// TwinCAT 3 PLC project EPS_Tests
// ProgramVersion: 3.1.4020.5
// libraries:
//   EPS, * (SLAC)
//   Tc2_BABasic, * (Beckhoff Automation GmbH)
//   Tc2_Standard, * (Beckhoff Automation GmbH)
//   Tc2_System, * (Beckhoff Automation GmbH)
//   Tc3_Module, * (Beckhoff Automation GmbH)
//   TcUnit, * (www.tcunit.org)
// project tree:
//   / PlcTask.TcTTO
//   POUs/Fixtures/AmphosMRC/ F_AmphosMRC_Error.TcPOU
//   POUs/Fixtures/BaseplateChiller/ F_BaseplateChiller_Error.TcPOU
//   POUs/Fixtures/DumpChiller/ F_DumpChiller_Error.TcPOU
//   POUs/Fixtures/Laser/ F_Laser_Error.TcPOU, F_LaserSetpoints.TcPOU
//   POUs/Fixtures/ChillerLoop/ F_ChillerLoop_Error.TcPOU
//   POUs/Fixtures/LeakMonitor/ F_LeakBoundaries.TcPOU, F_LeakMonitor_LIR_1.TcPOU, F_LeakMonitor_LIR_2.TcPOU, F_LeakMonitor_LOCO_2.TcPOU, F_LeakMonitor_LOTAO_2.TcPOU, F_LeakMonitor_LOTNL_1.TcPOU, F_LeakMonitor_LOTAO_1.TcPOU, F_LeakMonitor_LOCO_1.TcPOU, F_LeakMonitor_LOTNL_2.TcPOU, F_LeakMonitor_LUT_1.TcPOU, F_LeakMonitor_LUT_2.TcPOU
//   POUs/Fixtures/TemperatureMonitor/ F_TemperatureMonitorSetpoints.TcPOU, F_TemperatureMonitor_Error.TcPOU
//   POUs/ MAIN.TcPOU
//   POUs/TestSuites/UnitTests/Devices/ FB_AmphosMRC_Test.TcPOU, FB_BaseplateChiller_Test.TcPOU, FB_ChillerLoop_Test.TcPOU, FB_DumpChiller_Test.TcPOU, FB_Laser_Test.TcPOU, FB_LeakMonitor_Test.TcPOU, FB_TemperatureMonitor_Test.TcPOU
//   POUs/TestSuites/UnitTests/Interlocks/ FB_AmphosAttenuatorEnable_Test.TcPOU, FB_AmphosEnable_Test.TcPOU, FB_AmphosShutterEnable_Test.TcPOU, FB_BaseplateChillerEnable_Test.TcPOU, FB_CarbideShutterEnable_Test.TcPOU, FB_DumpChillerEnable_Test.TcPOU
// real-time tasks:
//   TASK PlcTask: cycle T#10ms, priority 20, ADS port 350

CONFIGURATION EPS_Tests
    RESOURCE PLC ON TwinCAT3
        TASK PlcTask(INTERVAL := T#10ms, PRIORITY := 20);
        PROGRAM MAIN WITH PlcTask : MAIN;
    END_RESOURCE
END_CONFIGURATION

// ---- POUs/MAIN.TcPOU
PROGRAM MAIN
VAR
	// Devices
	fbLeakMonitorTest : FB_LeakMonitor_Test;
	fbLoopTemperatureTest : FB_ChillerLoop_Test;
	fbLaserTest : FB_Laser_Test;
	fbTemperatureMonitorTest : FB_TemperatureMonitor_Test;
	fbDumpChillerTest : FB_DumpChiller_Test;
	fbBaseplateChillerTest : FB_BaseplateChiller_Test;
	fbAmphosMRCTest : FB_AmphosMRC_Test;
	
	// Interlocks
	fbAmphosAttenuatorEnableTest : FB_AmphosAttenuatorEnable_Test;
	fbAmphosShutterEnableTest : FB_AmphosShutterEnable_Test;
	fbCarbideShutterEnableTest : FB_CarbideShutterEnable_Test;
	fbDumpChillerEnableTest : FB_DumpChillerEnable_Test;
	fbBaseplateChillerEnableTest : FB_BaseplateChillerEnable_Test;
	fbAmphosEnableTest : FB_AmphosEnable_Test;
END_VAR

TcUnit.RUN();

END_PROGRAM

// ---- POUs/TestSuites/UnitTests/Devices/FB_LeakMonitor_Test.TcPOU
{attribute 'call_after_init'}
FUNCTION_BLOCK FB_LeakMonitor_Test EXTENDS FB_TestSuite
VAR_INPUT
END_VAR
VAR_OUTPUT
END_VAR
VAR
END_VAR

LOTAOTriggers1();
LOTAOTriggers2();
LOTAOLatches();
LOTAOResets();
LOTNLTriggers1();
LOTNLTriggers2();
LOTNLLatches();
LOTNLResets();
LOCOTriggers1();
LOCOTriggers2();
LOCOLatches();
LOCOResets();
LUTTriggers1();
LUTTriggers2();
LUTLatches();
LUTResets();
LIRTriggers1();
LIRTriggers2();
LIRLatches();
LIRResets();
NoLeak();

METHOD LIRLatches
VAR
	fbLeakMonitor : FB_LeakMonitor;
	stLeakBoundaries : ST_LeakBoundaries;
END_VAR
TEST('LeakInsideRacksLatches');

fbLeakMonitor := F_LeakMonitor_LIR_1(stBoundaries => stLeakBoundaries);

// Leak Error should stay latched even when inputs go back to normal
fbLeakMonitor(
	bLeakDetected := FALSE,
	stBound := stLeakBoundaries
);

AssertTrue(fbLeakMonitor.bLeakInsideRacks, 'Leak error did not stay latched');

TEST_FINISHED();
END_METHOD

METHOD LIRResets
VAR
	fbLeakMonitor : FB_LeakMonitor;
	stLeakBoundaries : ST_LeakBoundaries;
END_VAR
TEST('LeakInsideRacksResets');

fbLeakMonitor := F_LeakMonitor_LIR_1(stBoundaries => stLeakBoundaries);

// Error should be resettable
fbLeakMonitor.Reset();
fbLeakMonitor(bLeakDetected := FALSE, stBound := stLeakBoundaries);
AssertFalse(fbLeakMonitor.bLeakInsideRacks, 'Leak error did not reset');

TEST_FINISHED();
END_METHOD

METHOD LIRTriggers1
VAR
	fbLeakMonitor : FB_LeakMonitor := F_LeakMonitor_LIR_1();
END_VAR
TEST('LeakInsideRacksTriggers1');

AssertTrue(fbLeakMonitor.bLeakInsideRacks, 'Leak error did not trigger');

TEST_FINISHED();
END_METHOD

METHOD LIRTriggers2
VAR
	fbLeakMonitor : FB_LeakMonitor := F_LeakMonitor_LIR_2();
END_VAR
TEST('LeakInsideRacksTriggers2');

AssertTrue(fbLeakMonitor.bLeakInsideRacks, 'Leak error did not trigger');

TEST_FINISHED();
END_METHOD

METHOD LOCOLatches
VAR
	fbLeakMonitor : FB_LeakMonitor;
	stLeakBoundaries : ST_LeakBoundaries;
END_VAR
TEST('LeakOpcpaCarbideOnLatches');

fbLeakMonitor := F_LeakMonitor_LOCO_1(stBoundaries => stLeakBoundaries);

// Leak Error should stay latched even when inputs go back to normal
fbLeakMonitor(
	bLeakDetected := FALSE,
	stBound := stLeakBoundaries,
);
AssertTrue(fbLeakMonitor.bLeakOpcpaCarbideOn, 'Leak error did not stay latched');

TEST_FINISHED();
END_METHOD

METHOD LOCOResets
VAR
	fbLeakMonitor : FB_LeakMonitor;
	stLeakBoundaries : ST_LeakBoundaries;
END_VAR
TEST('LeakOpcpaCarbideOnResets');

fbLeakMonitor := F_LeakMonitor_LOCO_1(stBoundaries => stLeakBoundaries);

// Error should be resettable
fbLeakMonitor.Reset();
fbLeakMonitor(bLeakDetected := FALSE, stBound := stLeakBoundaries);
AssertFalse(fbLeakMonitor.bLeakOpcpaCarbideOn, 'Leak error did not reset');

TEST_FINISHED();
END_METHOD

METHOD LOCOTriggers1
VAR
	fbLeakMonitor : FB_LeakMonitor := F_LeakMonitor_LOCO_1();
END_VAR
TEST('LeakOpcpaCarbideOnTriggers11');

AssertTrue(fbLeakMonitor.bLeakOpcpaCarbideOn, 'Leak error did not trigger');

TEST_FINISHED();
END_METHOD

METHOD LOCOTriggers2
VAR
	fbLeakMonitor : FB_LeakMonitor := F_LeakMonitor_LOCO_2();
END_VAR
TEST('LeakOpcpaCarbideOnTriggers2');

AssertTrue(fbLeakMonitor.bLeakOpcpaCarbideOn, 'Leak error did not trigger');

TEST_FINISHED();
END_METHOD

METHOD LOTAOLatches
VAR
	fbLeakMonitor : FB_LeakMonitor;
	stLeakBoundaries : ST_LeakBoundaries;
END_VAR
TEST('LeakOpticalTableAmphosOnLatches');

fbLeakMonitor := F_LeakMonitor_LOTAO_1(stBoundaries => stLeakBoundaries);

// Leak Error should stay latched even when inputs go back to normal
fbLeakMonitor(
	bLeakDetected := FALSE,
	stBound := stLeakBoundaries
);

AssertTrue(fbLeakMonitor.bLeakOpticalTableAmphosOn, 'Leak error did not stay latched');

TEST_FINISHED();
END_METHOD

METHOD LOTAOResets
VAR
	fbLeakMonitor : FB_LeakMonitor;
	stLeakBoundaries : ST_LeakBoundaries;
END_VAR
TEST('LeakOpticalTableAmphosOnResets');

fbLeakMonitor := F_LeakMonitor_LOTAO_1(stBoundaries => stLeakBoundaries);

// Error should be resettable
fbLeakMonitor.Reset();
fbLeakMonitor(bLeakDetected := FALSE, stBound := stLeakBoundaries);
AssertFalse(fbLeakMonitor.bLeakOpticalTableAmphosOn, 'Leak error did not reset');

TEST_FINISHED();
END_METHOD

METHOD LOTAOTriggers1
VAR
	fbLeakMonitor : FB_LeakMonitor := F_LeakMonitor_LOTAO_1();
END_VAR
TEST('LeakOpticalTableAmphosOnTriggers1');

AssertTrue(fbLeakMonitor.bLeakOpticalTableAmphosOn, 'Leak error did not trigger');

TEST_FINISHED();
END_METHOD

METHOD LOTAOTriggers2
VAR
	fbLeakMonitor : FB_LeakMonitor := F_LeakMonitor_LOTAO_2();
END_VAR
TEST('LeakOpticalTableAmphosOnTriggers2');

AssertTrue(fbLeakMonitor.bLeakOpticalTableAmphosOn, 'Leak error did not trigger');

TEST_FINISHED();
END_METHOD

METHOD LOTNLLatches
VAR
	fbLeakMonitor : FB_LeakMonitor;
	stLeakBoundaries : ST_LeakBoundaries;
END_VAR
TEST('LeakOpticalTableNoLaserLatches');

fbLeakMonitor := F_LeakMonitor_LOTNL_1(stBoundaries => stLeakBoundaries);

// Leak Error should stay latched even when inputs go back to normal
fbLeakMonitor(
	bLeakDetected := FALSE,
	stBound := stLeakBoundaries
);
AssertTrue(fbLeakMonitor.bLeakOpticalTableNoLaser, 'Leak error did not stay latched');

TEST_FINISHED();
END_METHOD

METHOD LOTNLResets
VAR
	fbLeakMonitor : FB_LeakMonitor;
	stLeakBoundaries : ST_LeakBoundaries;
END_VAR
TEST('LeakOpticalTableNoLaserResets');

fbLeakMonitor := F_LeakMonitor_LOTNL_1(stBoundaries => stLeakBoundaries);

// Error should be resettable
fbLeakMonitor.Reset();
fbLeakMonitor(bLeakDetected := FALSE, stBound := stLeakBoundaries);
AssertFalse(fbLeakMonitor.bLeakOpticalTableNoLaser, 'Leak error did not reset');

TEST_FINISHED();
END_METHOD

METHOD LOTNLTriggers1
VAR
	fbLeakMonitor : FB_LeakMonitor := F_LeakMonitor_LOTNL_1();
END_VAR
TEST('LeakOpticalTableNoLaserTriggers1');

AssertTrue(fbLeakMonitor.bLeakOpticalTableNoLaser, 'Leak error did not trigger');

TEST_FINISHED();
END_METHOD

METHOD LOTNLTriggers2
VAR
	fbLeakMonitor : FB_LeakMonitor := F_LeakMonitor_LOTNL_2();
END_VAR
TEST('LeakOpticalTableNoLaserTriggers2');

AssertTrue(fbLeakMonitor.bLeakOpticalTableNoLaser, 'Leak error did not trigger');

TEST_FINISHED();
END_METHOD

METHOD LUTLatches
VAR
	fbLeakMonitor : FB_LeakMonitor;
	stLeakBoundaries : ST_LeakBoundaries;
END_VAR
TEST('LeakUnderTableLatches');

fbLeakMonitor := F_LeakMonitor_LUT_1(stBoundaries => stLeakBoundaries);

// Leak Error should stay latched even when inputs go back to normal
fbLeakMonitor(
	bLeakDetected := FALSE,
	stBound := stLeakBoundaries,
);
AssertTrue(fbLeakMonitor.bLeakUnderTable, 'Leak error did not stay latched');

TEST_FINISHED();
END_METHOD

METHOD LUTResets
VAR
	fbLeakMonitor : FB_LeakMonitor;
	stLeakBoundaries : ST_LeakBoundaries;
END_VAR
TEST('LeakUnderTableResets');

fbLeakMonitor := F_LeakMonitor_LUT_1(stBoundaries => stLeakBoundaries);

// Error should be resettable
fbLeakMonitor.Reset();
fbLeakMonitor(bLeakDetected := FALSE, stBound := stLeakBoundaries);
AssertFalse(fbLeakMonitor.bLeakUnderTable, 'Leak error did not reset');

TEST_FINISHED();
END_METHOD

METHOD LUTTriggers1
VAR
	fbLeakMonitor : FB_LeakMonitor := F_LeakMonitor_LUT_1();
END_VAR
TEST('LeakUnderTableTriggers1');

AssertTrue(fbLeakMonitor.bLeakUnderTable, 'Leak error did not trigger');

TEST_FINISHED();
END_METHOD

METHOD LUTTriggers2
VAR
	fbLeakMonitor : FB_LeakMonitor := F_LeakMonitor_LUT_2();
END_VAR
TEST('LeakUnderTableTriggers2');

AssertTrue(fbLeakMonitor.bLeakUnderTable, 'Leak error did not trigger');

TEST_FINISHED();
END_METHOD

METHOD NoLeak
VAR
	fbLeakMonitor : FB_LeakMonitor;
	stLeakBoundaries : ST_LeakBoundaries := F_LeakBoundaries();
END_VAR
TEST('NoLeak');

fbLeakMonitor(
	bLeakDetected := FALSE,
	bAmphosOn := TRUE,
	bCarbideOn := TRUE,
	stBound := stLeakBoundaries,
	nLocationResistance := stLeakBoundaries.nLMax6,
);
AssertFalse(fbLeakMonitor.bLeakOpticalTableAmphosOn OR fbLeakMonitor.bLeakOpticalTableNoLaser OR fbLeakMonitor.bLeakOpcpaCarbideOn OR fbLeakMonitor.bLeakUnderTable
	OR fbLeakMonitor.bLeakInsideRacks, 'Leak fasely detected');
	
TEST_FINISHED();
END_METHOD

END_FUNCTION_BLOCK

// ---- POUs/Fixtures/LeakMonitor/F_LeakMonitor_LIR_1.TcPOU
FUNCTION F_LeakMonitor_LIR_1 : FB_LeakMonitor
VAR_INPUT
END_VAR
VAR_OUTPUT
	// Provide stBoundaries output so test functions can reuse the boundaries
	stBoundaries : ST_LeakBoundaries := F_LeakBoundaries();
END_VAR
VAR
	fbLeakMonitor : FB_LeakMonitor;
END_VAR

fbLeakMonitor(
	bLeakDetected := TRUE,
	nLocationResistance := stBoundaries.nLMax6 - 1,
	stBound := stBoundaries
);

F_LeakMonitor_LIR_1 := fbLeakMonitor;

END_FUNCTION

// ---- POUs/Fixtures/LeakMonitor/F_LeakBoundaries.TcPOU
FUNCTION F_LeakBoundaries : ST_LeakBoundaries
VAR_INPUT
END_VAR
VAR
	stLeakBoundaries : ST_LeakBoundaries := (
		nLMin1 := 0,
		nLMax1 := 1000,
		nLMin2 := 1000,
		nLMax2 := 2000,
		nLMin3 := 2000,
		nLMax3 := 3000,
		nLMin4 := 3000,
		nLMax4 := 4000,
		nLMin5 := 4000,
		nLMax5 := 5000,
		nLMin6 := 5000,
		nLMax6 := 6000
	);
END_VAR

F_LeakBoundaries := stLeakBoundaries;

END_FUNCTION

// ---- POUs/Fixtures/LeakMonitor/F_LeakMonitor_LIR_2.TcPOU
FUNCTION F_LeakMonitor_LIR_2 : FB_LeakMonitor
VAR_INPUT
END_VAR
VAR_OUTPUT
	// Provide stBoundaries output so test functions can reuse the boundaries
	stBoundaries : ST_LeakBoundaries := F_LeakBoundaries();
END_VAR
VAR
	fbLeakMonitor : FB_LeakMonitor;
END_VAR

fbLeakMonitor(
	bLeakDetected := TRUE,
	nLocationResistance := stBoundaries.nLMin6,
	stBound := stBoundaries
);

F_LeakMonitor_LIR_2 := fbLeakMonitor;

END_FUNCTION

// ---- POUs/Fixtures/LeakMonitor/F_LeakMonitor_LOCO_1.TcPOU
FUNCTION F_LeakMonitor_LOCO_1 : FB_LeakMonitor
VAR_INPUT
END_VAR
VAR_OUTPUT
	// Provide stBoundaries output so test functions can reuse the boundaries
	stBoundaries : ST_LeakBoundaries := F_LeakBoundaries();
END_VAR
VAR
	fbLeakMonitor : FB_LeakMonitor;
END_VAR

fbLeakMonitor(
	bLeakDetected := TRUE,
	bCarbideOn := TRUE,
	nLocationResistance := stBoundaries.nLMax2 - 1,
	stBound := stBoundaries,
);

F_LeakMonitor_LOCO_1 := fbLeakMonitor;

END_FUNCTION

// ---- POUs/Fixtures/LeakMonitor/F_LeakMonitor_LOCO_2.TcPOU
FUNCTION F_LeakMonitor_LOCO_2 : FB_LeakMonitor
VAR_INPUT
END_VAR
VAR_OUTPUT
	// Provide stBoundaries output so test functions can reuse the boundaries
	stBoundaries : ST_LeakBoundaries := F_LeakBoundaries();
END_VAR
VAR
	fbLeakMonitor : FB_LeakMonitor;
END_VAR

fbLeakMonitor(
	bLeakDetected := TRUE,
	bCarbideOn := TRUE,
	nLocationResistance := stBoundaries.nLMin1,
	stBound := stBoundaries,
);

F_LeakMonitor_LOCO_2 := fbLeakMonitor;

END_FUNCTION

// ---- POUs/Fixtures/LeakMonitor/F_LeakMonitor_LOTAO_1.TcPOU
FUNCTION F_LeakMonitor_LOTAO_1 : FB_LeakMonitor
VAR_INPUT
END_VAR
VAR_OUTPUT
	// Provide stBoundaries output so test functions can reuse the boundaries
	stBoundaries : ST_LeakBoundaries := F_LeakBoundaries();
END_VAR
VAR
	fbLeakMonitor : FB_LeakMonitor;
END_VAR

fbLeakMonitor(
	bLeakDetected := TRUE,
	bAmphosOn := TRUE,
	nLocationResistance := stBoundaries.nLMax4 - 1,
	stBound := stBoundaries
);

F_LeakMonitor_LOTAO_1 := fbLeakMonitor;

END_FUNCTION

// ---- POUs/Fixtures/LeakMonitor/F_LeakMonitor_LOTAO_2.TcPOU
FUNCTION F_LeakMonitor_LOTAO_2 : FB_LeakMonitor
VAR_INPUT
END_VAR
VAR_OUTPUT
	// Provide stBoundaries output so test functions can reuse the boundaries
	stBoundaries : ST_LeakBoundaries := F_LeakBoundaries();
END_VAR
VAR
	fbLeakMonitor : FB_LeakMonitor;
END_VAR

fbLeakMonitor(
	bLeakDetected := TRUE,
	bAmphosOn := TRUE,
	nLocationResistance := stBoundaries.nLMin1,
	stBound := stBoundaries
);

F_LeakMonitor_LOTAO_2 := fbLeakMonitor;

END_FUNCTION

// ---- POUs/Fixtures/LeakMonitor/F_LeakMonitor_LOTNL_1.TcPOU
FUNCTION F_LeakMonitor_LOTNL_1 : FB_LeakMonitor
VAR_INPUT
END_VAR
VAR_OUTPUT
	// Provide stBoundaries output so test functions can reuse the boundaries
	stBoundaries : ST_LeakBoundaries := F_LeakBoundaries();
END_VAR
VAR
	fbLeakMonitor : FB_LeakMonitor;
END_VAR

fbLeakMonitor(
	bLeakDetected := TRUE,
	nLocationResistance := stBoundaries.nLMax4 - 1,
	stBound := stBoundaries,
);

F_LeakMonitor_LOTNL_1 := fbLeakMonitor;

END_FUNCTION

// ---- POUs/Fixtures/LeakMonitor/F_LeakMonitor_LOTNL_2.TcPOU
FUNCTION F_LeakMonitor_LOTNL_2 : FB_LeakMonitor
VAR_INPUT
END_VAR
VAR_OUTPUT
	// Provide stBoundaries output so test functions can reuse the boundaries
	stBoundaries : ST_LeakBoundaries := F_LeakBoundaries();
END_VAR
VAR
	fbLeakMonitor : FB_LeakMonitor;
END_VAR

fbLeakMonitor(
	bLeakDetected := TRUE,
	nLocationResistance := stBoundaries.nLMin1,
	stBound := stBoundaries,
);

F_LeakMonitor_LOTNL_2 := fbLeakMonitor;

END_FUNCTION

// ---- POUs/Fixtures/LeakMonitor/F_LeakMonitor_LUT_1.TcPOU
FUNCTION F_LeakMonitor_LUT_1 : FB_LeakMonitor
VAR_INPUT
END_VAR
VAR_OUTPUT
	// Provide stBoundaries output so test functions can reuse the boundaries
	stBoundaries : ST_LeakBoundaries := F_LeakBoundaries();
END_VAR
VAR
	fbLeakMonitor : FB_LeakMonitor;
END_VAR

fbLeakMonitor(
	bLeakDetected := TRUE,
	nLocationResistance := stBoundaries.nLMax5 -1,
	stBound := stBoundaries
);

F_LeakMonitor_LUT_1 := fbLeakMonitor;

END_FUNCTION

// ---- POUs/Fixtures/LeakMonitor/F_LeakMonitor_LUT_2.TcPOU
FUNCTION F_LeakMonitor_LUT_2 : FB_LeakMonitor
VAR_INPUT
END_VAR
VAR_OUTPUT
	// Provide stBoundaries output so test functions can reuse the boundaries
	stBoundaries : ST_LeakBoundaries := F_LeakBoundaries();
END_VAR
VAR
	fbLeakMonitor : FB_LeakMonitor;
END_VAR

fbLeakMonitor(
	bLeakDetected := TRUE,
	nLocationResistance := stBoundaries.nLMin5,
	stBound := stBoundaries
);

F_LeakMonitor_LUT_2 := fbLeakMonitor;

END_FUNCTION

// ---- POUs/TestSuites/UnitTests/Devices/FB_ChillerLoop_Test.TcPOU
{attribute 'call_after_init'}
FUNCTION_BLOCK FB_ChillerLoop_Test EXTENDS FB_TestSuite
VAR_INPUT
END_VAR
VAR_OUTPUT
END_VAR
VAR
END_VAR

TemperatureErrorTriggers();
TemperatureErrorReturnsToNormal();
NoError();
//OperatorOverrideResets();

METHOD NoError
VAR
	fbChillerLoop : FB_ChillerLoop;
END_VAR
TEST('NoChillerLoopError');

fbChillerLoop(bLoopTempSW := TRUE);
AssertFalse(fbChillerLoop.bError, 'Error fasely detected');

TEST_FINISHED();
END_METHOD

METHOD OperatorOverrideResets
VAR
	fbChillerLoop : FB_ChillerLoop;
END_VAR
(*
TEST('OperatorOverrideResets');

fbChillerLoop(bLoopTempSW := FALSE);
fbChillerLoop.bOperatorOverride := TRUE;
AssertTrue(fbChillerLoop.bOperatorOverride, 'Operator override failed to set');

// Operator override should reset uner normal temperature conditions.
fbChillerLoop(bLoopTempSW := TRUE);
AssertFalse(fbChillerLoop.bOperatorOverride, 'Operator override failed to reset');

TEST_FINISHED();
*)
END_METHOD

METHOD TemperatureErrorReturnsToNormal
VAR
	fbChillerLoop : FB_ChillerLoop := F_ChillerLoop_Error();
END_VAR
TEST('TemperatureErrorReturnsToNormal');

// Chiller loop should return to normal state when inputs go back to normal
fbChillerLoop(bLoopTempSW := TRUE);
AssertFalse(fbChillerLoop.bError, 'Temperature error did not go back to normal');

TEST_FINISHED();
END_METHOD

METHOD TemperatureErrorTriggers
VAR
	fbChillerLoop : FB_ChillerLoop := F_ChillerLoop_Error();
END_VAR
TEST('TemperatureErrorTriggers');

AssertTrue(fbChillerLoop.bError, 'Temperature error did not trigger');

TEST_FINISHED();
END_METHOD

END_FUNCTION_BLOCK

// ---- POUs/Fixtures/ChillerLoop/F_ChillerLoop_Error.TcPOU
FUNCTION F_ChillerLoop_Error : FB_ChillerLoop
VAR_INPUT
END_VAR
VAR
	fbChillerLoop : FB_ChillerLoop;
END_VAR

fbChillerLoop(bLoopTempSW := FALSE);
F_ChillerLoop_Error := fbChillerLoop;

END_FUNCTION

// ---- POUs/TestSuites/UnitTests/Devices/FB_Laser_Test.TcPOU
{attribute 'call_after_init'}
FUNCTION_BLOCK FB_Laser_Test EXTENDS FB_TestSuite
VAR_INPUT
END_VAR
VAR_OUTPUT
END_VAR
VAR
END_VAR

RawVoltageScales1();
RawVoltageScales2();
RawVoltageScales3();
LowVoltageTriggersError();
ErrorLatches();
ErrorResets();
NoError();

METHOD ErrorLatches
VAR
	fbLaser : FB_Laser;
	stSetpoints : ST_LaserSetpoints;
END_VAR
TEST('ErrorLatches');

// Trigger low voltage error
fbLaser := F_Laser_Error(stSetpoints => stSetpoints);

// Give non-erronuous input. Laser should stary latched
fbLaser(bAmphosOn := FALSE, stSetpoints := stSetpoints);
AssertTrue(fbLaser.bError, 'Laser did not stay latched');

TEST_FINISHED();
END_METHOD

METHOD ErrorResets
VAR
	fbLaser : FB_Laser;
	stSetpoints : ST_LaserSetpoints;
END_VAR
TEST('ErrorResets');

fbLaser := F_Laser_Error(stSetpoints => stSetpoints);

// Resetting the error on the laser should unlatch the system
fbLaser.Reset();
fbLaser(bAmphosOn := FALSE, stSetpoints := stSetpoints);
AssertFalse(fbLaser.bError, 'System did not unlatch when reset');

TEST_FINISHED();
END_METHOD

METHOD LowVoltageTriggersError
VAR
	fbLaser : FB_Laser := F_Laser_Error();
END_VAR
TEST('LowVoltageErrorTriggers');

AssertTrue(fbLaser.bError, 'Error not triggered');

TEST_FINISHED();
END_METHOD

METHOD NoError
VAR
	fbLaser : FB_Laser;
	stSetpoints : ST_LaserSetpoints := F_LaserSetpoints();
END_VAR
TEST('NoError');

fbLaser(
	nVoltageRaw := 16#7736,
	bAmphosOn := TRUE,
	stSetpoints := stSetpoints
);
AssertFalse(fbLaser.bError, 'Error fasely detected');

TEST_FINISHED();
END_METHOD

METHOD RawVoltageScales1
VAR
	fbLaser : FB_Laser;
	stSetpoints : ST_LaserSetpoints := F_LaserSetpoints();
END_VAR
TEST('RawVoltageScales1');

fbLaser(nVoltageRaw := 16#0000, stSetpoints := stSetpoints);
AssertEquals_LREAL(0, fbLaser.fVoltage, 0.01, 'Incorrect voltage scaling');

TEST_FINISHED();
END_METHOD

METHOD RawVoltageScales2
VAR
	fbLaser : FB_Laser;
	stSetpoints : ST_LaserSetpoints := F_LaserSetpoints();
END_VAR
TEST('RawVoltageScales2');

fbLaser(nVoltageRaw := 16#7736, stSetpoints := stSetpoints);
AssertEquals_LREAL(10, fbLaser.fVoltage, 0.01, 'Incorrect Amphos voltage scaling');

TEST_FINISHED();
END_METHOD

METHOD RawVoltageScales3
VAR
	fbLaser : FB_Laser;
	stSetpoints : ST_LaserSetpoints := F_LaserSetpoints();
END_VAR
TEST('RawVoltageScales3');

// Test behavior when given an overrange raw input
fbLaser(nVoltageRaw := 16#7FFF, stSetpoints := stSetpoints);
AssertEquals_LREAL(10, fbLaser.fVoltage, 0.01, 'Incorrect Amphos voltage scaling');

TEST_FINISHED();
END_METHOD

END_FUNCTION_BLOCK

// ---- POUs/Fixtures/Laser/F_Laser_Error.TcPOU
FUNCTION F_Laser_Error : FB_Laser
VAR_INPUT
END_VAR
VAR_OUTPUT
	stSetpoints : ST_LaserSetpoints := F_LaserSetpoints();
END_VAR
VAR
	fbLaser : FB_Laser;
END_VAR

fbLaser(
	nVoltageRaw := 0,
	bAmphosOn := TRUE,
	stSetpoints := stSetpoints
);

F_Laser_Error := fbLaser;

END_FUNCTION

// ---- POUs/Fixtures/Laser/F_LaserSetpoints.TcPOU
FUNCTION F_LaserSetpoints : ST_LaserSetpoints
VAR_INPUT
END_VAR
VAR
	stSetpoints : ST_LaserSetpoints := (
		nMinVoltage := 2,
		nMinNominalVoltage := 4
	);
END_VAR

F_LaserSetpoints := stSetpoints;

END_FUNCTION

// ---- POUs/TestSuites/UnitTests/Devices/FB_TemperatureMonitor_Test.TcPOU
{attribute 'call_after_init'}
FUNCTION_BLOCK FB_TemperatureMonitor_Test EXTENDS FB_TestSuite
VAR_INPUT
END_VAR
VAR_OUTPUT
END_VAR
VAR
END_VAR

ErrorTriggers();
ErrorGoesBackToNormal();
NoError();
TempMonRawScales1();
TempMonRawScales2();

METHOD ErrorGoesBackToNormal
VAR
	fbTempMon : FB_TemperatureMonitor;
	stSetpoints : ST_TemperatureMonitorSetpoints;
END_VAR
TEST('ErrorGoesBackToNormal');

// Error should go back to normal when temperature is in a safe range
fbTempMon := F_TemperatureMonitor_Error(stSetpoints => stSetpoints);
fbTempMon(nTempMonRaw := 0, stSetpoints := stSetpoints);
AssertFalse(fbTempMon.bError, 'Error did not go back to normal');

TEST_FINISHED();
END_METHOD

METHOD ErrorTriggers
VAR
	fbTempMon : FB_TemperatureMonitor := F_TemperatureMonitor_Error();
END_VAR
TEST('ErrorTriggers');

AssertTrue(fbTempMon.bError, 'Error did not trigger');
	
TEST_FINISHED();
END_METHOD

METHOD NoError
VAR
	fbTempMon : FB_TemperatureMonitor;
	stSetpoints : ST_TemperatureMonitorSetpoints := F_TemperatureMonitorSetpoints();
END_VAR
TEST('NoError');

fbTempMon(
	nTempMonRaw := 1, 
	bAmphosOn := TRUE, 
	stSetpoints := stSetpoints
);
AssertFalse(fbTempMon.bError, 'Error fasely detected');

TEST_FINISHED();
END_METHOD

METHOD TempMonRawScales1
VAR
	fbTempMon : FB_TemperatureMonitor;
	stSetpoints : ST_TemperatureMonitorSetpoints := F_TemperatureMonitorSetpoints();
END_VAR
TEST('TempMonRawScales1');

fbTempMon(
	nTempMonRaw := 0,
	stSetpoints := stSetpoints
);
AssertEquals_LREAL(0, fbTempMon.fTemperature, 0.01, 'Analog temperature scaling failed');

TEST_FINISHED();
END_METHOD

METHOD TempMonRawScales2
VAR
	fbTempMon : FB_TemperatureMonitor;
	stSetpoints : ST_TemperatureMonitorSetpoints := F_TemperatureMonitorSetpoints();
END_VAR
TEST('TempMonRawScales2');

fbTempMon(
	nTempMonRaw := 16#7736,
	stSetpoints := stSetpoints
);
AssertEquals_LREAL(1000, fbTempMon.fTemperature, 1, 'Analog temperature scaling failed');

TEST_FINISHED();
END_METHOD

END_FUNCTION_BLOCK

// ---- POUs/Fixtures/TemperatureMonitor/F_TemperatureMonitor_Error.TcPOU
FUNCTION F_TemperatureMonitor_Error : FB_TemperatureMonitor
VAR_INPUT
END_VAR
VAR_OUTPUT
	stSetpoints : ST_TemperatureMonitorSetpoints := F_TemperatureMonitorSetpoints();
END_VAR
VAR
	fbTempMon : FB_TemperatureMonitor;
END_VAR

fbTempMon(
	nTempMonRaw := 16#7736,
	bAmphosOn := TRUE,
	stSetpoints := stSetpoints
);
F_TemperatureMonitor_Error := fbTempMon;

END_FUNCTION

// ---- POUs/Fixtures/TemperatureMonitor/F_TemperatureMonitorSetpoints.TcPOU
FUNCTION F_TemperatureMonitorSetpoints : ST_TemperatureMonitorSetpoints
VAR_INPUT
END_VAR
VAR
	stTempMonSP : ST_TemperatureMonitorSetpoints := (fMaxTemperature := 40);
END_VAR

F_TemperatureMonitorSetpoints := stTempMonSP;

END_FUNCTION

// ---- POUs/TestSuites/UnitTests/Devices/FB_DumpChiller_Test.TcPOU
{attribute 'call_after_init'}
FUNCTION_BLOCK FB_DumpChiller_Test EXTENDS FB_TestSuite
VAR_INPUT
END_VAR
VAR_OUTPUT
END_VAR
VAR
END_VAR

ErrorTriggers();
ErrorResets();
ErrorLatches();
NoError();

METHOD ErrorLatches
VAR
	fbDumpChiller : FB_DumpChiller := F_DumpChiller_Error();
END_VAR
TEST('ErrorLatches');

fbDumpChiller(bDumpChillerFlow := TRUE);
AssertTrue(fbDumpChiller.bError, 'Error did not latch');

TEST_FINISHED();
END_METHOD

METHOD ErrorResets
VAR
	fbDumpChiller : FB_DumpChiller := F_DumpChiller_Error();
END_VAR
TEST('ErrorResets');

fbDumpChiller.Reset();
fbDumpChiller(bDumpChillerFlow := TRUE);
AssertFalse(fbDumpChiller.bError, 'Error did not reset');

TEST_FINISHED();
END_METHOD

METHOD ErrorTriggers
VAR
	fbDumpChiller : FB_DumpChiller := F_DumpChiller_Error();
END_VAR
TEST('ErrorTriggers');

AssertTrue(fbDumpChiller.bError, 'Error did not trigger');

TEST_FINISHED();
END_METHOD

METHOD NoError
VAR
	fbDumpChiller : FB_DumpChiller;
END_VAR
TEST('NoError');

fbDumpChiller(
	bAmphosOn := TRUE,
	bDumpChillerFlow := TRUE
);
AssertFalse(fbDumpChiller.bError, 'Error falsely triggered');

TEST_FINISHED();
END_METHOD

END_FUNCTION_BLOCK

// ---- POUs/Fixtures/DumpChiller/F_DumpChiller_Error.TcPOU
FUNCTION F_DumpChiller_Error : FB_DumpChiller
VAR_INPUT
END_VAR
VAR
	fbDumpChiller : FB_DumpChiller;
END_VAR

fbDumpChiller(
	bAmphosOn := TRUE,
	bDumpChillerFlow := FALSE
);
F_DumpChiller_Error := fbDumpChiller;

END_FUNCTION

// ---- POUs/TestSuites/UnitTests/Devices/FB_BaseplateChiller_Test.TcPOU
{attribute 'call_after_init'}
FUNCTION_BLOCK FB_BaseplateChiller_Test EXTENDS FB_TestSuite
VAR_INPUT
END_VAR
VAR_OUTPUT
END_VAR
VAR
END_VAR

ErrorTriggers();
ErrorResets();
ErrorLatches();
NoError();

METHOD ErrorLatches
VAR
	fbBaseplateChiller : FB_BaseplateChiller := F_BaseplateChiller_Error();
END_VAR
TEST('ErrorLatches');

fbBaseplateChiller(bBaseplateChillerFlow := TRUE);
AssertTrue(fbBaseplateChiller.bError, 'Error did not latch');

TEST_FINISHED();
END_METHOD

METHOD ErrorResets
VAR
	fbBaseplateChiller : FB_BaseplateChiller := F_BaseplateChiller_Error();
END_VAR
TEST('ErrorResets');

fbBaseplateChiller.Reset();
fbBaseplateChiller(bBaseplateChillerFlow := TRUE);
AssertFalse(fbBaseplateChiller.bError, 'Error did not reset');

TEST_FINISHED();
END_METHOD

METHOD ErrorTriggers
VAR
	fbBaseplateChiller : FB_BaseplateChiller := F_BaseplateChiller_Error();
END_VAR
TEST('ErrorTriggers');

AssertTrue(fbBaseplateChiller.bError, 'Error did not trigger');

TEST_FINISHED();
END_METHOD

METHOD NoError
VAR
	fbBaseplateChiller : FB_BaseplateChiller;
END_VAR
TEST('NoError');

fbBaseplateChiller(bBaseplateChillerFlow := TRUE);
AssertFalse(fbBaseplateChiller.bError, 'Error falsely triggered');

TEST_FINISHED();
END_METHOD

END_FUNCTION_BLOCK

// ---- POUs/Fixtures/BaseplateChiller/F_BaseplateChiller_Error.TcPOU
FUNCTION F_BaseplateChiller_Error : FB_BaseplateChiller
VAR_INPUT
END_VAR
VAR
	fbBaseplateChiller : FB_BaseplateChiller;
END_VAR

fbBaseplateChiller(bBaseplateChillerFlow := FALSE);
F_BaseplateChiller_Error := fbBaseplateChiller;

END_FUNCTION

// ---- POUs/TestSuites/UnitTests/Devices/FB_AmphosMRC_Test.TcPOU
{attribute 'call_after_init'}
FUNCTION_BLOCK FB_AmphosMRC_Test EXTENDS FB_TestSuite
VAR_INPUT
END_VAR
VAR_OUTPUT
END_VAR
VAR
END_VAR

ErrorTriggers();
ErrorGoesBackToNormal();
NoError();

METHOD ErrorGoesBackToNormal
VAR
	fbAmphosMRC : FB_AmphosMRC := F_AmphosMRC_Error();
END_VAR
TEST('ErrorGoesBackToNormal');

fbAmphosMRC(bMRC := TRUE);
AssertFalse(fbAmphosMRC.bError, 'Error did not go back to normal');

TEST_FINISHED();
END_METHOD

METHOD ErrorTriggers
VAR
	fbAmphosMRC : FB_AmphosMRC := F_AmphosMRC_Error();
END_VAR
TEST('ErrorTriggers');

AssertTrue(fbAmphosMRC.bError, 'Error did not trigger');

TEST_FINISHED();
END_METHOD

METHOD NoError
VAR
	fbAmphosMRC : FB_AmphosMRC;
END_VAR
TEST('NoError');

fbAmphosMRC(
	bAmphosOn := TRUE,
	bMRC := TRUE
);
AssertFalse(fbAmphosMRC.bError, 'Error falsely triggered');

TEST_FINISHED();
END_METHOD

END_FUNCTION_BLOCK

// ---- POUs/Fixtures/AmphosMRC/F_AmphosMRC_Error.TcPOU
FUNCTION F_AmphosMRC_Error : FB_AmphosMRC
VAR_INPUT
END_VAR
VAR
	fbAmphosMRC : FB_AmphosMRC;
END_VAR

fbAmphosMRC(
	bAmphosOn := TRUE,
	bMRC := FALSE
);
F_AmphosMRC_Error := fbAmphosMRC;

END_FUNCTION

// ---- POUs/TestSuites/UnitTests/Interlocks/FB_AmphosAttenuatorEnable_Test.TcPOU
{attribute 'call_after_init'}
FUNCTION_BLOCK FB_AmphosAttenuatorEnable_Test EXTENDS FB_TestSuite
VAR_INPUT
END_VAR
VAR_OUTPUT
END_VAR
VAR
END_VAR

LocksWithHardwareFailure();
LocksWithLUTLeak();
LocksWithLOTAOLeak();
LocksWithLOCOLeak();
LocksWithMRC01Error();
LocksWhenAmphosOff();
EnablesWhenNoError();

METHOD EnablesWhenNoError
VAR
	stErrors : st_ErrorStates;
	bResult : BOOL;
END_VAR
TEST('EnablesWhenNoError');

bResult := F_AmphosAttenuatorEnable(bAmphosOn := TRUE, stErrors := stErrors);

AssertTrue(bResult, 'Amphos Attenuator should be enabled');

TEST_FINISHED();
END_METHOD

METHOD LocksWhenAmphosOff
VAR
	stErrors : st_ErrorStates;
	bResult : BOOL;
END_VAR
TEST('LocksWhenAmphosOff');

bResult := F_AmphosAttenuatorEnable(bAmphosOn := FALSE, stErrors := stErrors);

AssertFalse(bResult, 'Amphos Attenuator did not lock');

TEST_FINISHED();
END_METHOD

METHOD LocksWithHardwareFailure
VAR
	stErrors : st_ErrorStates;
	bResult : BOOL;
END_VAR
TEST('LocksWithHardwareFailure');

stErrors.bHardwareFailure := TRUE;
bResult := F_AmphosAttenuatorEnable(bAmphosOn := FALSE, stErrors := stErrors);

AssertFalse(bResult, 'Amphos Attenuator did not lock');

TEST_FINISHED();
END_METHOD

METHOD LocksWithLOCOLeak
VAR
	stErrors : st_ErrorStates;
	bResult : BOOL;
END_VAR
TEST('LocksWithLOCOLeak');

stErrors.bLeakOpcpaCarbideOn := TRUE;
bResult := F_AmphosAttenuatorEnable(bAmphosOn := TRUE, stErrors := stErrors);

AssertFalse(bResult, 'Amphos Attenuator did not lock');

TEST_FINISHED();
END_METHOD

METHOD LocksWithLOTAOLeak
VAR
	stErrors : st_ErrorStates;
	bResult : BOOL;
END_VAR
TEST('LocksWithLOTAOLeak');

stErrors.bLeakOpticalTableAmphosOn := TRUE;
bResult := F_AmphosAttenuatorEnable(bAmphosOn := TRUE, stErrors := stErrors);

AssertFalse(bResult, 'Amphos Attenuator did not lock');

TEST_FINISHED();
END_METHOD

METHOD LocksWithLUTLeak
VAR
	stErrors : st_ErrorStates;
	bResult : BOOL;
END_VAR
TEST('LocksWithLUTLeak');

stErrors.bLeakUnderTable := TRUE;
bResult := F_AmphosAttenuatorEnable(bAmphosOn := TRUE, stErrors := stErrors);

AssertFalse(bResult, 'Amphos Attenuator did not lock');

TEST_FINISHED();
END_METHOD

METHOD LocksWithMRC01Error
VAR
	stErrors : st_ErrorStates;
	bResult : BOOL;
END_VAR
TEST('LocksWithMRC01Error');

stErrors.bAmphosMRC01 := TRUE;
bResult := F_AmphosAttenuatorEnable(bAmphosOn := TRUE, stErrors := stErrors);

AssertFalse(bResult, 'Amphos Attenuator did not lock');

TEST_FINISHED();
END_METHOD

END_FUNCTION_BLOCK

// ---- POUs/TestSuites/UnitTests/Interlocks/FB_AmphosShutterEnable_Test.TcPOU
{attribute 'call_after_init'}
FUNCTION_BLOCK FB_AmphosShutterEnable_Test EXTENDS FB_TestSuite
VAR_INPUT
END_VAR
VAR_OUTPUT
END_VAR
VAR
END_VAR

LocksWithHardwareFailure();
LocksWithLOCOLeak();
LocksWithLOTAOLeak();
LocksWithLUTLeak();
LocksWithAmphosOnAndTemperatureEvent01();
LocksWithAmphosOnAndTemperatureEvent02();
LocksWithAmphosOnAndTemperatureEvent03();
LocksWithAmphosOnAndTemperatureEvent04();
LocksWithTempMonError01();
LocksWithTempMonError02();
LocksWithTempMonError03();
LocksWithTempMonError04();
LocksWithTempMonError05();
LocksWithTempMonError06();
LocksWithTempMonError07();
LocksWithTempMonError08();
LocksWithOpcpaCriticalError();
LocksWithDumpChillerError();
LocksWithMRCError02();
LocksWithMRCError03();
EnablesWithAmphosOffAndTemperatureEvent01();
EnablesWithAmphosOffAndTemperatureEvent02();
EnablesWithAmphosOffAndTemperatureEvent03();
EnablesWithAmphosOffAndTemperatureEvent04();
EnablesWithTemperatureEventOverride01();
EnablesWithTemperatureEventOverride02();
EnablesWithTemperatureEventOverride03();
EnablesWithTemperatureEventOverride04();
EnablesWithOpcpaMinorError();
EnablesWhenNoError();

METHOD EnablesWhenNoError
VAR
	stErrors : st_ErrorStates;
	stOpcpaSetpoints : ST_LaserSetpoints := F_LaserSetpoints();
	bResult : BOOL;
END_VAR
TEST('EnablesWhenNoError');

bResult := F_AmphosShutterEnable(
	bAmphosOn := TRUE, 
	fOpcpaVoltage := stOpcpaSetpoints.nMinNominalVoltage, 
	bLoopTempOverride01 := FALSE,
	bLoopTempOverride02 := FALSE,
	bLoopTempOverride03 := FALSE,
	bLoopTempOverride04 := FALSE,
	stErrors := stErrors,
	stOpcpaSetpoints := stOpcpaSetpoints
);

AssertTrue(bResult, 'Amphos Shutter did not enable');

TEST_FINISHED();
END_METHOD

METHOD EnablesWithAmphosOffAndTemperatureEvent01
VAR
	stErrors : st_ErrorStates;
	stOpcpaSetpoints : ST_LaserSetpoints := F_LaserSetpoints();
	bResult : BOOL;
END_VAR
TEST('EnablesWithAmphosOffAndTemperatureEvent01');

stErrors.bChillerLoop01 := TRUE;
bResult := F_AmphosShutterEnable(
	bAmphosOn := FALSE, 
	fOpcpaVoltage := stOpcpaSetpoints.nMinNominalVoltage, 
	bLoopTempOverride01 := FALSE,
	bLoopTempOverride02 := FALSE,
	bLoopTempOverride03 := FALSE,
	bLoopTempOverride04 := FALSE,
	stErrors := stErrors,
	stOpcpaSetpoints := stOpcpaSetpoints
);

AssertTrue(bResult, 'Amphos Shutter did not enable');

TEST_FINISHED();
END_METHOD

METHOD EnablesWithAmphosOffAndTemperatureEvent02
VAR
	stErrors : st_ErrorStates;
	stOpcpaSetpoints : ST_LaserSetpoints := F_LaserSetpoints();
	bResult : BOOL;
END_VAR
TEST('EnablesWithAmphosOffAndTemperatureEvent02');

stErrors.bChillerLoop02 := TRUE;
bResult := F_AmphosShutterEnable(
	bAmphosOn := FALSE, 
	fOpcpaVoltage := stOpcpaSetpoints.nMinNominalVoltage, 
	bLoopTempOverride01 := FALSE,
	bLoopTempOverride02 := FALSE,
	bLoopTempOverride03 := FALSE,
	bLoopTempOverride04 := FALSE,
	stErrors := stErrors,
	stOpcpaSetpoints := stOpcpaSetpoints
);

AssertTrue(bResult, 'Amphos Shutter did not enable');

TEST_FINISHED();
END_METHOD

METHOD EnablesWithAmphosOffAndTemperatureEvent03
VAR
	stErrors : st_ErrorStates;
	stOpcpaSetpoints : ST_LaserSetpoints := F_LaserSetpoints();
	bResult : BOOL;
END_VAR
TEST('EnablesWithAmphosOffAndTemperatureEvent03');

stErrors.bChillerLoop03 := TRUE;
bResult := F_AmphosShutterEnable(
	bAmphosOn := FALSE, 
	fOpcpaVoltage := stOpcpaSetpoints.nMinNominalVoltage, 
	bLoopTempOverride01 := FALSE,
	bLoopTempOverride02 := FALSE,
	bLoopTempOverride03 := FALSE,
	bLoopTempOverride04 := FALSE,
	stErrors := stErrors,
	stOpcpaSetpoints := stOpcpaSetpoints
);

AssertTrue(bResult, 'Amphos Shutter did not enable');

TEST_FINISHED();
END_METHOD

METHOD EnablesWithAmphosOffAndTemperatureEvent04
VAR
	stErrors : st_ErrorStates;
	stOpcpaSetpoints : ST_LaserSetpoints := F_LaserSetpoints();
	bResult : BOOL;
END_VAR
TEST('EnablesWithAmphosOffAndTemperatureEvent04');

stErrors.bChillerLoop04 := TRUE;
bResult := F_AmphosShutterEnable(
	bAmphosOn := FALSE, 
	fOpcpaVoltage := stOpcpaSetpoints.nMinNominalVoltage, 
	bLoopTempOverride01 := FALSE,
	bLoopTempOverride02 := FALSE,
	bLoopTempOverride03 := FALSE,
	bLoopTempOverride04 := FALSE,
	stErrors := stErrors,
	stOpcpaSetpoints := stOpcpaSetpoints
);

AssertTrue(bResult, 'Amphos Shutter did not enable');

TEST_FINISHED();
END_METHOD

METHOD EnablesWithOpcpaMinorError
VAR
	stErrors : st_ErrorStates;
	stOpcpaSetpoints : ST_LaserSetpoints := F_LaserSetpoints();
	bResult : BOOL;
END_VAR
TEST('EnablesWithOpcpaMinorError');

stErrors.bOpcpaBeam := TRUE;
bResult := F_AmphosShutterEnable(
	bAmphosOn := TRUE, 
	fOpcpaVoltage := stOpcpaSetpoints.nMinNominalVoltage - 0.001, 
	bLoopTempOverride01 := FALSE,
	bLoopTempOverride02 := FALSE,
	bLoopTempOverride03 := FALSE,
	bLoopTempOverride04 := FALSE,
	stErrors := stErrors,
	stOpcpaSetpoints := stOpcpaSetpoints
);

AssertTrue(bResult, 'Amphos Shutter did not enable');

TEST_FINISHED();
END_METHOD

METHOD EnablesWithTemperatureEventOverride01
VAR
	stErrors : st_ErrorStates;
	stOpcpaSetpoints : ST_LaserSetpoints := F_LaserSetpoints();
	bResult : BOOL;
END_VAR
TEST('EnablesWithTemperatureEventOverride01');

stErrors.bChillerLoop01 := TRUE;
bResult := F_AmphosShutterEnable(
	bAmphosOn := TRUE, 
	fOpcpaVoltage := stOpcpaSetpoints.nMinNominalVoltage, 
	bLoopTempOverride01 := TRUE,
	bLoopTempOverride02 := FALSE,
	bLoopTempOverride03 := FALSE,
	bLoopTempOverride04 := FALSE,
	stErrors := stErrors,
	stOpcpaSetpoints := stOpcpaSetpoints
);

AssertTrue(bResult, 'Amphos Shutter did not enable');

TEST_FINISHED();
END_METHOD

METHOD EnablesWithTemperatureEventOverride02
VAR
	stErrors : st_ErrorStates;
	stOpcpaSetpoints : ST_LaserSetpoints := F_LaserSetpoints();
	bResult : BOOL;
END_VAR
TEST('EnablesWithTemperatureEventOverride02');

stErrors.bChillerLoop02 := TRUE;
bResult := F_AmphosShutterEnable(
	bAmphosOn := TRUE, 
	fOpcpaVoltage := stOpcpaSetpoints.nMinNominalVoltage, 
	bLoopTempOverride01 := FALSE,
	bLoopTempOverride02 := TRUE,
	bLoopTempOverride03 := FALSE,
	bLoopTempOverride04 := FALSE,
	stErrors := stErrors,
	stOpcpaSetpoints := stOpcpaSetpoints
);

AssertTrue(bResult, 'Amphos Shutter did not enable');

TEST_FINISHED();
END_METHOD

METHOD EnablesWithTemperatureEventOverride03
VAR
	stErrors : st_ErrorStates;
	stOpcpaSetpoints : ST_LaserSetpoints := F_LaserSetpoints();
	bResult : BOOL;
END_VAR
TEST('EnablesWithTemperatureEventOverride03');

stErrors.bChillerLoop03 := TRUE;
bResult := F_AmphosShutterEnable(
	bAmphosOn := TRUE, 
	fOpcpaVoltage := stOpcpaSetpoints.nMinNominalVoltage, 
	bLoopTempOverride01 := FALSE,
	bLoopTempOverride02 := FALSE,
	bLoopTempOverride03 := TRUE,
	bLoopTempOverride04 := FALSE,
	stErrors := stErrors,
	stOpcpaSetpoints := stOpcpaSetpoints
);

AssertTrue(bResult, 'Amphos Shutter did not enable');

TEST_FINISHED();
END_METHOD

METHOD EnablesWithTemperatureEventOverride04
VAR
	stErrors : st_ErrorStates;
	stOpcpaSetpoints : ST_LaserSetpoints := F_LaserSetpoints();
	bResult : BOOL;
END_VAR
TEST('EnablesWithTemperatureEventOverride04');

stErrors.bChillerLoop04 := TRUE;
bResult := F_AmphosShutterEnable(
	bAmphosOn := TRUE, 
	fOpcpaVoltage := stOpcpaSetpoints.nMinNominalVoltage, 
	bLoopTempOverride01 := FALSE,
	bLoopTempOverride02 := FALSE,
	bLoopTempOverride03 := FALSE,
	bLoopTempOverride04 := TRUE,
	stErrors := stErrors,
	stOpcpaSetpoints := stOpcpaSetpoints
);

AssertTrue(bResult, 'Amphos Shutter did not enable');

TEST_FINISHED();
END_METHOD

METHOD LocksWithAmphosOnAndTemperatureEvent01
VAR
	stErrors : st_ErrorStates;
	stOpcpaSetpoints : ST_LaserSetpoints := F_LaserSetpoints();
	bResult : BOOL;
END_VAR
TEST('LocksWithAmphosOnAndTemperatureEvent01');

stErrors.bChillerLoop01 := TRUE;
bResult := F_AmphosShutterEnable(
	bAmphosOn := TRUE, 
	fOpcpaVoltage := stOpcpaSetpoints.nMinNominalVoltage, 
	bLoopTempOverride01 := FALSE,
	bLoopTempOverride02 := FALSE,
	bLoopTempOverride03 := FALSE,
	bLoopTempOverride04 := FALSE,
	stErrors := stErrors,
	stOpcpaSetpoints := stOpcpaSetpoints
);

AssertFalse(bResult, 'Amphos Shutter did not lock');

TEST_FINISHED();
END_METHOD

METHOD LocksWithAmphosOnAndTemperatureEvent02
VAR
	stErrors : st_ErrorStates;
	stOpcpaSetpoints : ST_LaserSetpoints := F_LaserSetpoints();
	bResult : BOOL;
END_VAR
TEST('LocksWithAmphosOnAndTemperatureEvent02');

stErrors.bChillerLoop02 := TRUE;
bResult := F_AmphosShutterEnable(
	bAmphosOn := TRUE, 
	fOpcpaVoltage := stOpcpaSetpoints.nMinNominalVoltage, 
	bLoopTempOverride01 := FALSE,
	bLoopTempOverride02 := FALSE,
	bLoopTempOverride03 := FALSE,
	bLoopTempOverride04 := FALSE,
	stErrors := stErrors,
	stOpcpaSetpoints := stOpcpaSetpoints
);

AssertFalse(bResult, 'Amphos Shutter did not lock');

TEST_FINISHED();
END_METHOD

METHOD LocksWithAmphosOnAndTemperatureEvent03
VAR
	stErrors : st_ErrorStates;
	stOpcpaSetpoints : ST_LaserSetpoints := F_LaserSetpoints();
	bResult : BOOL;
END_VAR
TEST('LocksWithAmphosOnAndTemperatureEvent03');

stErrors.bChillerLoop03 := TRUE;
bResult := F_AmphosShutterEnable(
	bAmphosOn := TRUE, 
	fOpcpaVoltage := stOpcpaSetpoints.nMinNominalVoltage, 
	bLoopTempOverride01 := FALSE,
	bLoopTempOverride02 := FALSE,
	bLoopTempOverride03 := FALSE,
	bLoopTempOverride04 := FALSE,
	stErrors := stErrors,
	stOpcpaSetpoints := stOpcpaSetpoints
);

AssertFalse(bResult, 'Amphos Shutter did not lock');

TEST_FINISHED();
END_METHOD

METHOD LocksWithAmphosOnAndTemperatureEvent04
VAR
	stErrors : st_ErrorStates;
	stOpcpaSetpoints : ST_LaserSetpoints := F_LaserSetpoints();
	bResult : BOOL;
END_VAR
TEST('LocksWithAmphosOnAndTemperatureEvent04');

stErrors.bChillerLoop04 := TRUE;
bResult := F_AmphosShutterEnable(
	bAmphosOn := TRUE, 
	fOpcpaVoltage := stOpcpaSetpoints.nMinNominalVoltage, 
	bLoopTempOverride01 := FALSE,
	bLoopTempOverride02 := FALSE,
	bLoopTempOverride03 := FALSE,
	bLoopTempOverride04 := FALSE,
	stErrors := stErrors,
	stOpcpaSetpoints := stOpcpaSetpoints
);

AssertFalse(bResult, 'Amphos Shutter did not lock');

TEST_FINISHED();
END_METHOD

METHOD LocksWithDumpChillerError
VAR
	stErrors : st_ErrorStates;
	stOpcpaSetpoints : ST_LaserSetpoints := F_LaserSetpoints();
	bResult : BOOL;
END_VAR
TEST('LocksWithDumpChillerError');

stErrors.bDumpChiller := TRUE;
bResult := F_AmphosShutterEnable(
	bAmphosOn := TRUE, 
	fOpcpaVoltage := stOpcpaSetpoints.nMinNominalVoltage, 
	bLoopTempOverride01 := FALSE,
	bLoopTempOverride02 := FALSE,
	bLoopTempOverride03 := FALSE,
	bLoopTempOverride04 := FALSE,
	stErrors := stErrors,
	stOpcpaSetpoints := stOpcpaSetpoints
);

AssertFalse(bResult, 'Amphos Shutter did not lock');

TEST_FINISHED();
END_METHOD

METHOD LocksWithHardwareFailure
VAR
	stErrors : st_ErrorStates;
	stOpcpaSetpoints : ST_LaserSetpoints := F_LaserSetpoints();
	bResult : BOOL;
END_VAR
TEST('LocksWithHardwareFailure');

stErrors.bHardwareFailure := TRUE;
bResult := F_AmphosShutterEnable(
	bAmphosOn := TRUE, 
	fOpcpaVoltage := stOpcpaSetpoints.nMinNominalVoltage, 
	bLoopTempOverride01 := FALSE,
	bLoopTempOverride02 := FALSE,
	bLoopTempOverride03 := FALSE,
	bLoopTempOverride04 := FALSE,
	stErrors := stErrors,
	stOpcpaSetpoints := stOpcpaSetpoints
);

AssertFalse(bResult, 'Amphos Shutter did not lock');

TEST_FINISHED();
END_METHOD

METHOD LocksWithLOCOLeak
VAR
	stErrors : st_ErrorStates;
	stOpcpaSetpoints : ST_LaserSetpoints := F_LaserSetpoints();
	bResult : BOOL;
END_VAR
TEST('LocksWithLOCOLeak');

stErrors.bLeakOpcpaCarbideOn := TRUE;
bResult := F_AmphosShutterEnable(
	bAmphosOn := TRUE, 
	fOpcpaVoltage := stOpcpaSetpoints.nMinNominalVoltage, 
	bLoopTempOverride01 := FALSE,
	bLoopTempOverride02 := FALSE,
	bLoopTempOverride03 := FALSE,
	bLoopTempOverride04 := FALSE,
	stErrors := stErrors,
	stOpcpaSetpoints := stOpcpaSetpoints
);

AssertFalse(bResult, 'Amphos Shutter did not lock');

TEST_FINISHED();
END_METHOD

METHOD LocksWithLOTAOLeak
VAR
	stErrors : st_ErrorStates;
	stOpcpaSetpoints : ST_LaserSetpoints := F_LaserSetpoints();
	bResult : BOOL;
END_VAR
TEST('LocksWithLOTAOLeak');

stErrors.bLeakOpticalTableAmphosOn := TRUE;
bResult := F_AmphosShutterEnable(
	bAmphosOn := TRUE, 
	fOpcpaVoltage := stOpcpaSetpoints.nMinNominalVoltage, 
	bLoopTempOverride01 := FALSE,
	bLoopTempOverride02 := FALSE,
	bLoopTempOverride03 := FALSE,
	bLoopTempOverride04 := FALSE,
	stErrors := stErrors,
	stOpcpaSetpoints := stOpcpaSetpoints
);

AssertFalse(bResult, 'Amphos Shutter did not lock');

TEST_FINISHED();
END_METHOD

METHOD LocksWithLUTLeak
VAR
	stErrors : st_ErrorStates;
	stOpcpaSetpoints : ST_LaserSetpoints := F_LaserSetpoints();
	bResult : BOOL;
END_VAR
TEST('LocksWithLUTLeak');

stErrors.bLeakUnderTable := TRUE;
bResult := F_AmphosShutterEnable(
	bAmphosOn := TRUE, 
	fOpcpaVoltage := stOpcpaSetpoints.nMinNominalVoltage, 
	bLoopTempOverride01 := FALSE,
	bLoopTempOverride02 := FALSE,
	bLoopTempOverride03 := FALSE,
	bLoopTempOverride04 := FALSE,
	stErrors := stErrors,
	stOpcpaSetpoints := stOpcpaSetpoints
);

AssertFalse(bResult, 'Amphos Shutter did not lock');

TEST_FINISHED();
END_METHOD

METHOD LocksWithMRCError02
VAR
	stErrors : st_ErrorStates;
	stOpcpaSetpoints : ST_LaserSetpoints := F_LaserSetpoints();
	bResult : BOOL;
END_VAR
TEST('LocksWithMRCError02');

stErrors.bAmphosMRC02 := TRUE;
bResult := F_AmphosShutterEnable(
	bAmphosOn := TRUE, 
	fOpcpaVoltage := stOpcpaSetpoints.nMinNominalVoltage, 
	bLoopTempOverride01 := FALSE,
	bLoopTempOverride02 := FALSE,
	bLoopTempOverride03 := FALSE,
	bLoopTempOverride04 := FALSE,
	stErrors := stErrors,
	stOpcpaSetpoints := stOpcpaSetpoints
);

AssertFalse(bResult, 'Amphos Shutter did not lock');

TEST_FINISHED();
END_METHOD

METHOD LocksWithMRCError03
VAR
	stErrors : st_ErrorStates;
	stOpcpaSetpoints : ST_LaserSetpoints := F_LaserSetpoints();
	bResult : BOOL;
END_VAR
TEST('LocksWithMRCError03');

stErrors.bAmphosMRC03 := TRUE;
bResult := F_AmphosShutterEnable(
	bAmphosOn := TRUE, 
	fOpcpaVoltage := stOpcpaSetpoints.nMinNominalVoltage, 
	bLoopTempOverride01 := FALSE,
	bLoopTempOverride02 := FALSE,
	bLoopTempOverride03 := FALSE,
	bLoopTempOverride04 := FALSE,
	stErrors := stErrors,
	stOpcpaSetpoints := stOpcpaSetpoints
);

AssertFalse(bResult, 'Amphos Shutter did not lock');

TEST_FINISHED();
END_METHOD

METHOD LocksWithOpcpaCriticalError
VAR
	stErrors : st_ErrorStates;
	stOpcpaSetpoints : ST_LaserSetpoints := F_LaserSetpoints();
	bResult : BOOL;
END_VAR
TEST('LocksWithOpcpaCriticalError');

stErrors.bOpcpaBeam := TRUE;
bResult := F_AmphosShutterEnable(
	bAmphosOn := TRUE, 
	fOpcpaVoltage := stOpcpaSetpoints.nMinVoltage - 1, 
	bLoopTempOverride01 := FALSE,
	bLoopTempOverride02 := FALSE,
	bLoopTempOverride03 := FALSE,
	bLoopTempOverride04 := FALSE,
	stErrors := stErrors,
	stOpcpaSetpoints := stOpcpaSetpoints
);

AssertFalse(bResult, 'Amphos Shutter did not lock');

TEST_FINISHED();
END_METHOD

METHOD LocksWithTempMonError01
VAR
	stErrors : st_ErrorStates;
	stOpcpaSetpoints : ST_LaserSetpoints := F_LaserSetpoints();
	bResult : BOOL;
END_VAR
TEST('LocksWithTempMonError01');

stErrors.bTempMon01 := TRUE;
bResult := F_AmphosShutterEnable(
	bAmphosOn := TRUE, 
	fOpcpaVoltage := stOpcpaSetpoints.nMinNominalVoltage, 
	bLoopTempOverride01 := FALSE,
	bLoopTempOverride02 := FALSE,
	bLoopTempOverride03 := FALSE,
	bLoopTempOverride04 := FALSE,
	stErrors := stErrors,
	stOpcpaSetpoints := stOpcpaSetpoints
);

AssertFalse(bResult, 'Amphos Shutter did not lock');

TEST_FINISHED();
END_METHOD

METHOD LocksWithTempMonError02
VAR
	stErrors : st_ErrorStates;
	stOpcpaSetpoints : ST_LaserSetpoints := F_LaserSetpoints();
	bResult : BOOL;
END_VAR
TEST('LocksWithTempMonError02');

stErrors.bTempMon02 := TRUE;
bResult := F_AmphosShutterEnable(
	bAmphosOn := TRUE, 
	fOpcpaVoltage := stOpcpaSetpoints.nMinNominalVoltage, 
	bLoopTempOverride01 := FALSE,
	bLoopTempOverride02 := FALSE,
	bLoopTempOverride03 := FALSE,
	bLoopTempOverride04 := FALSE,
	stErrors := stErrors,
	stOpcpaSetpoints := stOpcpaSetpoints
);

AssertFalse(bResult, 'Amphos Shutter did not lock');

TEST_FINISHED();
END_METHOD

METHOD LocksWithTempMonError03
VAR
	stErrors : st_ErrorStates;
	stOpcpaSetpoints : ST_LaserSetpoints := F_LaserSetpoints();
	bResult : BOOL;
END_VAR
TEST('LocksWithTempMonError03');

stErrors.bTempMon03 := TRUE;
bResult := F_AmphosShutterEnable(
	bAmphosOn := TRUE, 
	fOpcpaVoltage := stOpcpaSetpoints.nMinNominalVoltage, 
	bLoopTempOverride01 := FALSE,
	bLoopTempOverride02 := FALSE,
	bLoopTempOverride03 := FALSE,
	bLoopTempOverride04 := FALSE,
	stErrors := stErrors,
	stOpcpaSetpoints := stOpcpaSetpoints
);

AssertFalse(bResult, 'Amphos Shutter did not lock');

TEST_FINISHED();
END_METHOD

METHOD LocksWithTempMonError04
VAR
	stErrors : st_ErrorStates;
	stOpcpaSetpoints : ST_LaserSetpoints := F_LaserSetpoints();
	bResult : BOOL;
END_VAR
TEST('LocksWithTempMonError04');

stErrors.bTempMon04 := TRUE;
bResult := F_AmphosShutterEnable(
	bAmphosOn := TRUE, 
	fOpcpaVoltage := stOpcpaSetpoints.nMinNominalVoltage, 
	bLoopTempOverride01 := FALSE,
	bLoopTempOverride02 := FALSE,
	bLoopTempOverride03 := FALSE,
	bLoopTempOverride04 := FALSE,
	stErrors := stErrors,
	stOpcpaSetpoints := stOpcpaSetpoints
);

AssertFalse(bResult, 'Amphos Shutter did not lock');

TEST_FINISHED();
END_METHOD

METHOD LocksWithTempMonError05
VAR
	stErrors : st_ErrorStates;
	stOpcpaSetpoints : ST_LaserSetpoints := F_LaserSetpoints();
	bResult : BOOL;
END_VAR
TEST('LocksWithTempMonError05');

stErrors.bTempMon05 := TRUE;
bResult := F_AmphosShutterEnable(
	bAmphosOn := TRUE, 
	fOpcpaVoltage := stOpcpaSetpoints.nMinNominalVoltage, 
	bLoopTempOverride01 := FALSE,
	bLoopTempOverride02 := FALSE,
	bLoopTempOverride03 := FALSE,
	bLoopTempOverride04 := FALSE,
	stErrors := stErrors,
	stOpcpaSetpoints := stOpcpaSetpoints
);

AssertFalse(bResult, 'Amphos Shutter did not lock');

TEST_FINISHED();
END_METHOD

METHOD LocksWithTempMonError06
VAR
	stErrors : st_ErrorStates;
	stOpcpaSetpoints : ST_LaserSetpoints := F_LaserSetpoints();
	bResult : BOOL;
END_VAR
TEST('LocksWithTempMonError06');

stErrors.bTempMon06 := TRUE;
bResult := F_AmphosShutterEnable(
	bAmphosOn := TRUE, 
	fOpcpaVoltage := stOpcpaSetpoints.nMinNominalVoltage, 
	bLoopTempOverride01 := FALSE,
	bLoopTempOverride02 := FALSE,
	bLoopTempOverride03 := FALSE,
	bLoopTempOverride04 := FALSE,
	stErrors := stErrors,
	stOpcpaSetpoints := stOpcpaSetpoints
);

AssertFalse(bResult, 'Amphos Shutter did not lock');

TEST_FINISHED();
END_METHOD

METHOD LocksWithTempMonError07
VAR
	stErrors : st_ErrorStates;
	stOpcpaSetpoints : ST_LaserSetpoints := F_LaserSetpoints();
	bResult : BOOL;
END_VAR
TEST('LocksWithTempMonError07');

stErrors.bTempMon07 := TRUE;
bResult := F_AmphosShutterEnable(
	bAmphosOn := TRUE, 
	fOpcpaVoltage := stOpcpaSetpoints.nMinNominalVoltage, 
	bLoopTempOverride01 := FALSE,
	bLoopTempOverride02 := FALSE,
	bLoopTempOverride03 := FALSE,
	bLoopTempOverride04 := FALSE,
	stErrors := stErrors,
	stOpcpaSetpoints := stOpcpaSetpoints
);

AssertFalse(bResult, 'Amphos Shutter did not lock');

TEST_FINISHED();
END_METHOD

METHOD LocksWithTempMonError08
VAR
	stErrors : st_ErrorStates;
	stOpcpaSetpoints : ST_LaserSetpoints := F_LaserSetpoints();
	bResult : BOOL;
END_VAR
TEST('LocksWithTempMonError08');

stErrors.bTempMon08 := TRUE;
bResult := F_AmphosShutterEnable(
	bAmphosOn := TRUE, 
	fOpcpaVoltage := stOpcpaSetpoints.nMinNominalVoltage, 
	bLoopTempOverride01 := FALSE,
	bLoopTempOverride02 := FALSE,
	bLoopTempOverride03 := FALSE,
	bLoopTempOverride04 := FALSE,
	stErrors := stErrors,
	stOpcpaSetpoints := stOpcpaSetpoints
);

AssertFalse(bResult, 'Amphos Shutter did not lock');

TEST_FINISHED();
END_METHOD

END_FUNCTION_BLOCK

// ---- POUs/TestSuites/UnitTests/Interlocks/FB_CarbideShutterEnable_Test.TcPOU
{attribute 'call_after_init'}
FUNCTION_BLOCK FB_CarbideShutterEnable_Test EXTENDS FB_TestSuite
VAR_INPUT
END_VAR
VAR_OUTPUT
END_VAR
VAR
END_VAR

LocksWithHardwareFailure();
LocksWithLOCOLeak();
LocksWithLUTLeak();
EnablesWhenNoError();

METHOD EnablesWhenNoError
VAR
	stErrors : ST_ErrorStates;
	bResult : BOOL;
END_VAR
TEST('EnablesWhenNoErrors');

bResult := F_CarbideShutterEnable(stErrors := stErrors);

AssertTrue(bResult, 'Carbide Shutter did not enable');

TEST_FINISHED();
END_METHOD

METHOD LocksWithHardwareFailure
VAR
	stErrors : st_ErrorStates;
	bResult : BOOL;
END_VAR
TEST('LocksWithHardwareFailure');

stErrors.bHardwareFailure := TRUE;
bResult := F_CarbideShutterEnable(stErrors := stErrors);

AssertFalse(bResult, 'Carbide Shutter did not lock');

TEST_FINISHED();
END_METHOD

METHOD LocksWithLOCOLeak
VAR
	stErrors : st_ErrorStates;
	bResult : BOOL;
END_VAR
TEST('LocksWithLOCOLeak');

stErrors.bLeakOpcpaCarbideOn := TRUE;
bResult := F_CarbideShutterEnable(stErrors := stErrors);

AssertFalse(bResult, 'Carbide Shutter did not lock');

TEST_FINISHED();
END_METHOD

METHOD LocksWithLUTLeak
VAR
	stErrors : st_ErrorStates;
	bResult : BOOL;
END_VAR
TEST('LocksWithLUTLeak');

stErrors.bLeakUnderTable := TRUE;
bResult := F_CarbideShutterEnable(stErrors := stErrors);

AssertFalse(bResult, 'Carbide Shutter did not lock');

TEST_FINISHED();
END_METHOD

END_FUNCTION_BLOCK

// ---- POUs/TestSuites/UnitTests/Interlocks/FB_DumpChillerEnable_Test.TcPOU
{attribute 'call_after_init'}
FUNCTION_BLOCK FB_DumpChillerEnable_Test EXTENDS FB_TestSuite
VAR_INPUT
END_VAR
VAR_OUTPUT
END_VAR
VAR
END_VAR

LocksWithHardwareFailure();
LocksWithLUTLeak();
LocksWithLOTAOLeak();
LocksWithLOTNLLeak();
LocksWithLOCOLeak();
EnablesWhenNoError();

METHOD EnablesWhenNoError
VAR
	stErrors : st_ErrorStates;
	bResult : BOOL;
END_VAR
TEST('EnablesWhenNoError');

bResult := F_DumpChillerEnable(stErrors := stErrors);

AssertTrue(bResult, 'Dump chiller relay did not close');

TEST_FINISHED();
END_METHOD

METHOD LocksWithHardwareFailure
VAR
	stErrors : st_ErrorStates;
	bResult : BOOL;
END_VAR
TEST('LocksWithHardwareFailure');

stErrors.bHardwareFailure := TRUE;
bResult := F_DumpChillerEnable(stErrors := stErrors);

AssertFalse(bResult, 'Dump chiller relay did not open');

TEST_FINISHED();
END_METHOD

METHOD LocksWithLOCOLeak
VAR
	stErrors : st_ErrorStates;
	bResult : BOOL;
END_VAR
TEST('LocksWithLOCOLeak');

stErrors.bLeakOpcpaCarbideOn := TRUE;
bResult := F_DumpChillerEnable(stErrors := stErrors);

AssertFalse(bResult, 'Dump chiller relay did not open');

TEST_FINISHED();
END_METHOD

METHOD LocksWithLOTAOLeak
VAR
	stErrors : st_ErrorStates;
	bResult : BOOL;
END_VAR
TEST('LocksWithLOTAOLeak');

stErrors.bLeakOpticalTableAmphosOn := TRUE;
bResult := F_DumpChillerEnable(stErrors := stErrors);

AssertFalse(bResult, 'Dump chiller relay did not open');

TEST_FINISHED();
END_METHOD

METHOD LocksWithLOTNLLeak
VAR
	stErrors : st_ErrorStates;
	bResult : BOOL;
END_VAR
TEST('LocksWithLOTNLLeak');

stErrors.bLeakOpticalTableNoLaser := TRUE;
bResult := F_DumpChillerEnable(stErrors := stErrors);

AssertFalse(bResult, 'Dump chiller relay did not open');

TEST_FINISHED();
END_METHOD

METHOD LocksWithLUTLeak
VAR
	stErrors : st_ErrorStates;
	bResult : BOOL;
END_VAR
TEST('LocksWithLUTLeak');

stErrors.bLeakUnderTable := TRUE;
bResult := F_DumpChillerEnable(stErrors := stErrors);

AssertFalse(bResult, 'Dump chiller relay did not open');

TEST_FINISHED();
END_METHOD

END_FUNCTION_BLOCK

// ---- POUs/TestSuites/UnitTests/Interlocks/FB_BaseplateChillerEnable_Test.TcPOU
{attribute 'call_after_init'}
FUNCTION_BLOCK FB_BaseplateChillerEnable_Test EXTENDS FB_TestSuite
VAR_INPUT
END_VAR
VAR_OUTPUT
END_VAR
VAR
END_VAR

LocksWithHardwareFailure();
LocksWithLUTLeak();
EnablesWhenNoError();

METHOD EnablesWhenNoError
VAR
	stErrors : st_ErrorStates;
	bResult : BOOL;
END_VAR
TEST('EnablesWhenNoError');

bResult := F_BaseplateChillerEnable(stErrors := stErrors);

AssertTrue(bResult, 'Baseplate chiller relay did not close');

TEST_FINISHED();
END_METHOD

METHOD LocksWithHardwareFailure
VAR
	stErrors : st_ErrorStates;
	bResult : BOOL;
END_VAR
TEST('LocksWithHardwareFailure');

stErrors.bHardwareFailure := TRUE;
bResult := F_BaseplateChillerEnable(stErrors := stErrors);

AssertFalse(bResult, 'Baseplate chiller relay did not open');

TEST_FINISHED();
END_METHOD

METHOD LocksWithLUTLeak
VAR
	stErrors : st_ErrorStates;
	bResult : BOOL;
END_VAR
TEST('LocksWithLUTLeak');

stErrors.bLeakUnderTable := TRUE;
bResult := F_BaseplateChillerEnable(stErrors := stErrors);

AssertFalse(bResult, 'Baseplate chiller relay did not open');

TEST_FINISHED();
END_METHOD

END_FUNCTION_BLOCK

// ---- POUs/TestSuites/UnitTests/Interlocks/FB_AmphosEnable_Test.TcPOU
{attribute 'call_after_init'}
FUNCTION_BLOCK FB_AmphosEnable_Test EXTENDS FB_TestSuite
VAR_INPUT
END_VAR
VAR_OUTPUT
END_VAR
VAR
END_VAR

LocksWithHardwareFailure();
EnablesWithAmphosMinorError();
LocksWithAmphosCriticalError();
EnablesWhenNoError();
LocksWithPrevError();
UnlocksWithBeamErrorReset();

METHOD EnablesWhenNoError
VAR
	stErrors : st_ErrorStates;
	stAmphosSetpoints : ST_LaserSetpoints := F_LaserSetpoints();
	bResult : BOOL;
END_VAR
TEST('EnablesWhenNoError');

bResult := F_AmphosEnable(
	fAmphosVoltage := stAmphosSetpoints.nMinNominalVoltage,
	bEnabled := TRUE,
	stAmphosSetpoints := stAmphosSetpoints,
	stErrors := stErrors
);
AssertTrue(bResult, 'Amphos did not enable');

TEST_FINISHED();
END_METHOD

METHOD EnablesWithAmphosMinorError
VAR
	stErrors : st_ErrorStates;
	stAmphosSetpoints : ST_LaserSetpoints := F_LaserSetpoints();
	bResult : BOOL;
END_VAR
TEST('EnablesWithAmphosMinorError');

stErrors.bAmphosBeam := TRUE;
bResult := F_AmphosEnable(
	fAmphosVoltage := stAmphosSetpoints.nMinNominalVoltage - 0.001,
	bEnabled := TRUE,
	stAmphosSetpoints := stAmphosSetpoints,
	stErrors := stErrors
);
AssertTrue(bResult, 'Amphos did not enable');

TEST_FINISHED();
END_METHOD

METHOD LocksWithAmphosCriticalError
VAR
	stErrors : st_ErrorStates;
	stAmphosSetpoints : ST_LaserSetpoints := F_LaserSetpoints();
	bResult : BOOL;
END_VAR
TEST('LocksWithAmphosCriticalError');

stErrors.bAmphosBeam := TRUE;
bResult := F_AmphosEnable(
	fAmphosVoltage := stAmphosSetpoints.nMinVoltage - 0.1,
	bEnabled := TRUE,
	stAmphosSetpoints := stAmphosSetpoints,
	stErrors := stErrors
);
AssertFalse(bResult, 'Amphos did not lock');

TEST_FINISHED();
END_METHOD

METHOD LocksWithHardwareFailure
VAR
	stErrors : st_ErrorStates;
	stAmphosSetpoints : ST_LaserSetpoints := F_LaserSetpoints();
	bResult : BOOL;
END_VAR
TEST('LocksWithHardwareFailure');

stErrors.bHardwareFailure := TRUE;
bResult := F_AmphosEnable(
	fAmphosVoltage := stAmphosSetpoints.nMinNominalVoltage,
	bEnabled := TRUE,
	stAmphosSetpoints := stAmphosSetpoints,
	stErrors := stErrors
);
AssertFalse(bResult, 'Amphos did not lock');

TEST_FINISHED();
END_METHOD

METHOD LocksWithPrevError
VAR
	stErrors : st_ErrorStates;
	stAmphosSetpoints : ST_LaserSetpoints := F_LaserSetpoints();
	bResult : BOOL;
END_VAR
TEST('LatchesWithAmphosCriticalError');

// If the interlock previously failed and there is still a beam error, then lock and stay locked until beam error reset, even if there is only a minor error
stErrors.bAmphosBeam := TRUE;
bResult := F_AmphosEnable(
	fAmphosVoltage := stAmphosSetpoints.nMinNominalVoltage - 0.001, // Minor error
	bEnabled := FALSE,
	stAmphosSetpoints := stAmphosSetpoints,
	stErrors := stErrors
);
AssertFalse(bResult, 'Amphos did not lock');

TEST_FINISHED();
END_METHOD

METHOD UnlocksWithBeamErrorReset
VAR
	stErrors : st_ErrorStates;
	stAmphosSetpoints : ST_LaserSetpoints := F_LaserSetpoints();
	bResult : BOOL;
END_VAR
TEST('Unlocks with beam error reset');

// Even if bEnabled was false last time, reset if the beam error is now cleared
bResult := F_AmphosEnable(
	fAmphosVoltage := stAmphosSetpoints.nMinNominalVoltage,
	bEnabled := FALSE,
	stAmphosSetpoints := stAmphosSetpoints,
	stErrors := stErrors
);
AssertTrue(bResult, 'Amphos did not enable');

TEST_FINISHED();
END_METHOD

END_FUNCTION_BLOCK
